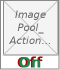
VISUALIZATION Plug  // 60x70
VAR_IN_OUT
	Etat_MaAr	:BOOL;
END_VAR
    Rectangle (0,55 60x15), "Off", invisible if: Etat_MaAr, text list: 'OuvFerm', text index: S_Cmd_ElectroValve_Alim_Lavabo
    Rectangle (0,55 60x15), "On", invisible if: NOT Etat_MaAr, text list: 'OuvFerm', text index: S_Cmd_ElectroValve_Alim_Lavabo
    Image (3,0 55x55), invisible if: Etat_MaAr, image: ImagePool_Action.Plug_Offe
    Image (3,0 55x55), invisible if: NOT Etat_MaAr, image: ImagePool_Action.Plug_On
END_VISUALIZATION

(* stored: Version 1.1.0.1, ProductVersion 3.1.4024.15
   Visu Plug: Id {77b1f7a7-9542-46bf-9b34-30ef8588e9d8} *)
